FUNCTION_BLOCK ALR2_TO_ALR (* Composite FB for convert bidirectional ALR2 to unidirectional ALR *)
  (* Standard: 61499-2; Function: ALR2_BIDIR forwards its incoming (EO1) side out as a plain unidirectional signal via ALR_OUT. ALR_IN publishes its value onto the outgoing (EI1) side of ALR2_BIDIR.; Description: Copyright (c) 2026 HR Agrartechnik GmbH This program and the accompanying materials are made available under the terms of the Eclipse Public License 2.0 which is available at https://www.eclipse.org/legal/epl-2.0/ SPDX-License-Identifier: EPL-2.0 *)
  (* Version 1.0, 2026-09-12, Franz Höpfinger, HR Agrartechnik GmbH, Initial Version - Konvertierungsfamilie vervollstaendigt (analog zu AR2/AB2/AE2). *)
  PACKAGE adapter::conversion::bidirectional;
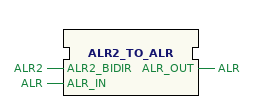
  SOCKETS
    ALR2_BIDIR : adapter::types::bidirectional::ALR2; (* Adapter Input: bidirectional tap, incoming side forwarded to ALR_OUT, outgoing side driven by ALR_IN *)
    ALR_IN : adapter::types::unidirectional::ALR; (* Adapter Input: unidirectional source *)
  END_SOCKETS
  PLUGS
    ALR_OUT : adapter::types::unidirectional::ALR; (* Adapter Output: mirrors ALR2_BIDIR's incoming (indication) side *)
  END_PLUGS
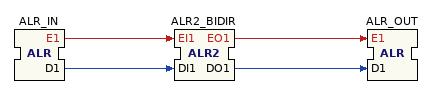
  EVENT_CONNECTIONS
    ALR2_BIDIR.EO1 TO ALR_OUT.E1;
    ALR_IN.E1 TO ALR2_BIDIR.EI1;
  END_CONNECTIONS
  DATA_CONNECTIONS
    ALR2_BIDIR.DO1 TO ALR_OUT.D1;
    ALR_IN.D1 TO ALR2_BIDIR.DI1;
  END_CONNECTIONS
END_FUNCTION_BLOCK
